PROGRAM MAIN
VAR
	m : INT;
END_VAR

m := m + 1;
PrgMqttCom();

END_PROGRAM

(* stored: Version 1.1.0.1, ProductVersion 3.1.4022.18
   POU MAIN: Id {a00b47c4-e886-489a-8899-d512157aae0f}, SpecialFunc None *)
